FUNCTION F_CalculateThicknessFromTransmission : LREAL
(*
    Thickness returned in units of meters.
    Negative result means invalid input.
    Absorption constant must be greater than 0.
    Transmission must be between 0.0 and 1.0 inclusive.
*)
VAR_INPUT
    fAbsorptionConstant : LREAL; (* The absorption constant mu, calculated by F_CalculateXrayAbsorptionConstant *)
    fTransmission : LREAL; (* Transmission to get thickness for [unitless] *)
END_VAR


IF fAbsorptionConstant <= 0 OR fTransmission < 0.0 OR fTransmission > 1.0 THEN
    F_CalculateThicknessFromTransmission := -1.0;
    RETURN;
END_IF

F_CalculateThicknessFromTransmission := LN(fTransmission) / -fAbsorptionConstant;

END_FUNCTION

(* stored: Version 1.1.0.1
   POU F_CalculateThicknessFromTransmission: Id {86ab3c10-17a1-4a58-9757-d4465e13dde9}, SpecialFunc None *)
